PROGRAM slave
VAR
END_VAR

END_PROGRAM

(* stored: Version 1.1.0.1, ProductVersion 3.1.4024.4
   POU slave: Id {45ef1047-11b4-4376-af2d-d1048d98e90e}, SpecialFunc None *)
